(* CODESYS project TrabalhoFinal.project

Project tree, tasks and I/O mapping:
  Device : CODESYS Control Win V3, 3S - Smart Software Solutions GmbH, order no. 305021, version 3.5.11.30
    application Application
      libraries: Standard, * (System); Util, * (System)
      task MainTask (cyclic, interval t#20ms, priority 1) calls PLC_PRG
      program PLC_PRG [LD]
      Symbols
*)

// Device/Application/PLC_PRG
PROGRAM PLC_PRG
VAR
	_PassaCaixa: BOOL;
	_AtBack:BOOL;
	_AtEntry:BOOL;
	_AtFront:BOOL;
	_AtLeftEntry:BOOL;
	_AtLeftExit:BOOL;
	_AtLoadPosition:BOOL;
	_AtRigthEntry:BOOL;
	_AtRigthExit:BOOL;
	_AtTurnableEntry:BOOL;
	_AtUnloadPosition:BOOL;
	_Auto:BOOL;
	_EmergencyStop:BOOL;
	_HighBox:BOOL;
	_LowBox:BOOL;
	_Pallet:BOOL;
	_Manual:BOOL;
	_Resert:BOOL;
	_Start:BOOL;
	_Stop:BOOL;

	EntryConveyor:BOOL;
	FeederConveyor:BOOL;
	GreenIndicator:BOOL;
	LeftConveyor:BOOL;
	Load:BOOL;
	RedIndicator:BOOL;
	ResetLigth:BOOL;
	RightConveyor:BOOL;
	StartLigth:BOOL;
	StopLigth:BOOL;
	Turn:BOOL;
	Unload:BOOL;
	YellowIndicator:BOOL;
	ShortBox:BOOL;
	HighBox:BOOL;
	Trig_Right_Entry : F_TRIG;
	Trig_Left_Exit : F_TRIG;
	Trig_Rigth_Exit : F_TRIG;
	Trig_Mov1 : R_TRIG;
	Trig_Mov2 : R_TRIG;
	Trig_Mov3 : R_TRIG;
	Trig_Mov4 : R_TRIG;
	Trig_Mov5 : R_TRIG;
	Trig_turnable_Entry : F_TRIG;
	aux: INT;
	aux1:INT;
	aux2:INT;
	aux3:INT;
	auxMov1: BOOL;
	auxMov2: BOOL;
	auxMov3: BOOL;
	TON_0: TON;
	TON_1: TON;
	VarTimer1: TIME;
	VarTimer2: TIME;
	VarTimer3: TIME;
	Descarrega:BOOL;
	carregaAtivaLoad: BOOL;
	descarregaAtivaLoad: BOOL;
	descarregaAtivaUnload: BOOL;
	R_TRIG_0: R_TRIG;
	resetAux:bool;
	F_TRIG_0: F_TRIG;
	F_TRIG_1: F_TRIG;
	F_TRIG_2: F_TRIG;
	TON_2: TON;
	aux4: INT;
	ativadorTurn:BOOL;
	CTU_0: CTU;
	resetContadores: BOOL;
	contCaixasTotal:int;
	CTU_1: CTU;
	contCaixaAltas: INT;
	contCaixaBaixas: INT;
	F_TRIG_3: F_TRIG;
	F_TRIG_4: F_TRIG;
	F_TRIG_5: F_TRIG;
	
	para_esteira_principal:BOOL;
	
	sup_ligar:BOOL;
	sup_desligar:BOOL;
	sup_emergencia:BOOL;
	sup_reset:BOOL;

	sup_pos_rota:INT;
	
	
	R_TRIG_1: R_TRIG;
END_VAR
VAR // added by the converter: edge detectors and wires of the graphical bodies
    _w1, _w2, _w3, _w4, _w5 : BOOL;
END_VAR

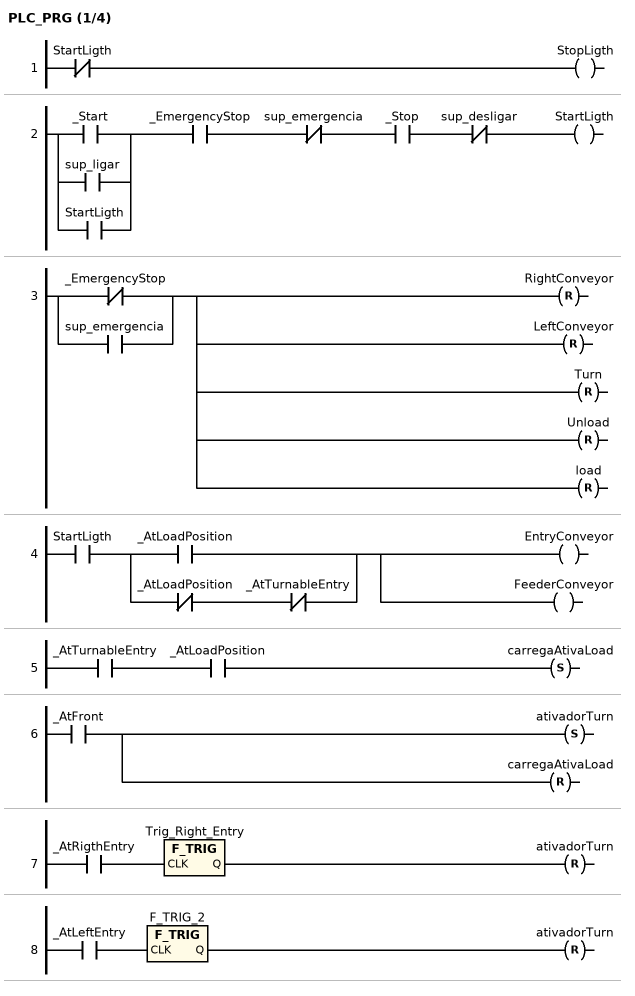
// NETWORK 1
StopLigth := NOT StartLigth;

// NETWORK 2
StartLigth := (_Start OR sup_ligar OR StartLigth) AND _EmergencyStop AND NOT sup_emergencia AND _Stop AND NOT sup_desligar;

// NETWORK 3
_w1 := NOT _EmergencyStop OR sup_emergencia;
RightConveyor R= _w1;
LeftConveyor R= _w1;
Turn R= _w1;
Unload R= _w1;
load R= _w1;

// NETWORK 4
_w2 := StartLigth AND (_AtLoadPosition OR NOT _AtLoadPosition AND NOT _AtTurnableEntry);
EntryConveyor := _w2;
FeederConveyor := _w2;

// NETWORK 5
carregaAtivaLoad S= _AtTurnableEntry AND _AtLoadPosition;

// NETWORK 6
ativadorTurn S= _AtFront;
carregaAtivaLoad R= _AtFront;

// NETWORK 7
Trig_Right_Entry(CLK := _AtRigthEntry); // F_TRIG
ativadorTurn R= Trig_Right_Entry.Q;

// NETWORK 8
F_TRIG_2(CLK := _AtLeftEntry); // F_TRIG
ativadorTurn R= F_TRIG_2.Q;

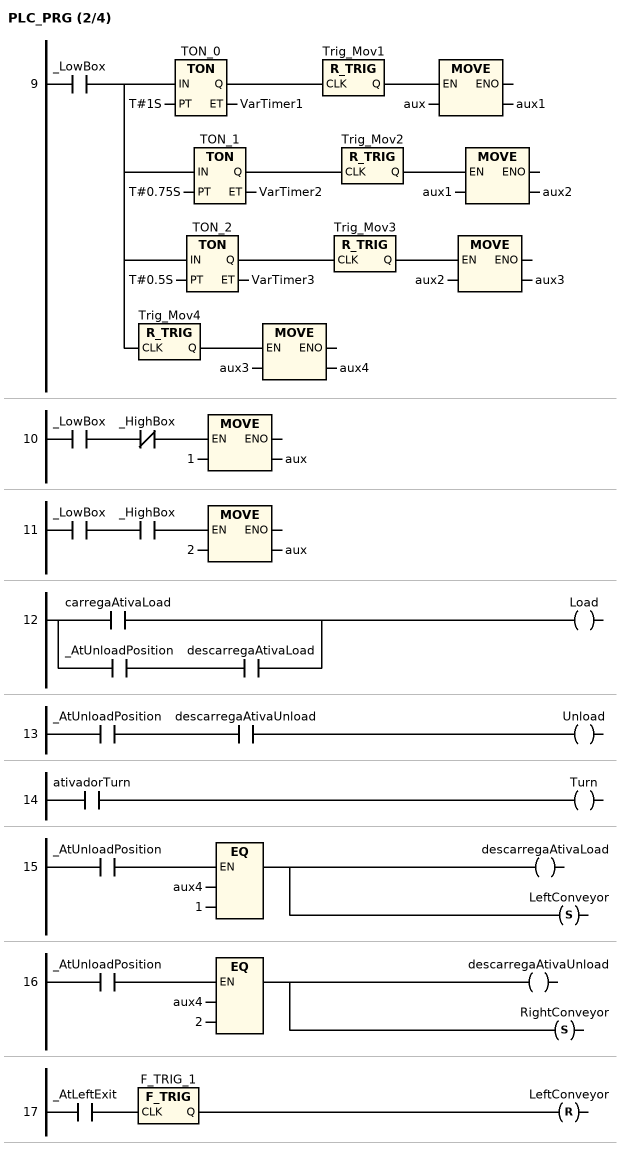
// NETWORK 9
TON_0(IN := _LowBox, PT := T#1S, ET => VarTimer1); // TON
Trig_Mov1(CLK := TON_0.Q); // R_TRIG
IF Trig_Mov1.Q THEN aux1 := aux; END_IF
TON_1(IN := _LowBox, PT := T#0.75S, ET => VarTimer2); // TON
Trig_Mov2(CLK := TON_1.Q); // R_TRIG
IF Trig_Mov2.Q THEN aux2 := aux1; END_IF
TON_2(IN := _LowBox, PT := T#0.5S, ET => VarTimer3); // TON
Trig_Mov3(CLK := TON_2.Q); // R_TRIG
IF Trig_Mov3.Q THEN aux3 := aux2; END_IF
Trig_Mov4(CLK := _LowBox); // R_TRIG
IF Trig_Mov4.Q THEN aux4 := aux3; END_IF

// NETWORK 10
IF _LowBox AND NOT _HighBox THEN aux := 1; END_IF

// NETWORK 11
IF _LowBox AND _HighBox THEN aux := 2; END_IF

// NETWORK 12
Load := carregaAtivaLoad OR _AtUnloadPosition AND descarregaAtivaLoad;

// NETWORK 13
Unload := _AtUnloadPosition AND descarregaAtivaUnload;

// NETWORK 14
Turn := ativadorTurn;

// NETWORK 15
_w3 := _AtUnloadPosition AND aux4 = 1;
descarregaAtivaLoad := _w3;
LeftConveyor S= _w3;

// NETWORK 16
_w4 := _AtUnloadPosition AND aux4 = 2;
descarregaAtivaUnload := _w4;
RightConveyor S= _w4;

// NETWORK 17
F_TRIG_1(CLK := _AtLeftExit); // F_TRIG
LeftConveyor R= F_TRIG_1.Q;

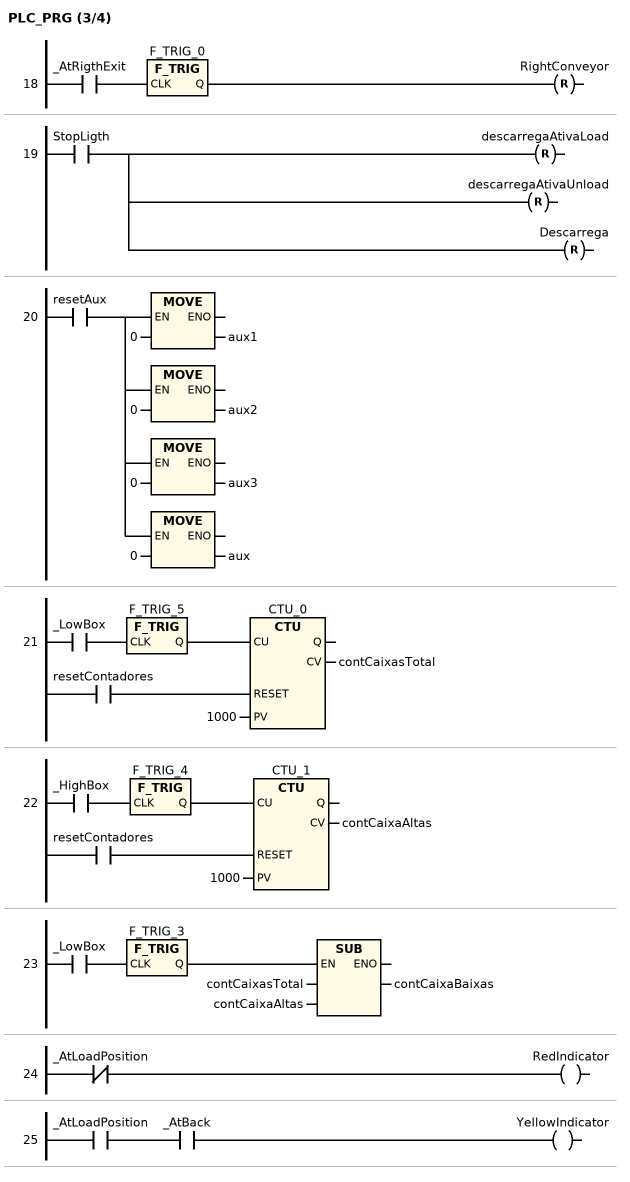
// NETWORK 18
F_TRIG_0(CLK := _AtRigthExit); // F_TRIG
RightConveyor R= F_TRIG_0.Q;

// NETWORK 19
descarregaAtivaLoad R= StopLigth;
descarregaAtivaUnload R= StopLigth;
Descarrega R= StopLigth;

// NETWORK 20
IF resetAux THEN aux1 := 0; END_IF
IF resetAux THEN aux2 := 0; END_IF
IF resetAux THEN aux3 := 0; END_IF
IF resetAux THEN aux := 0; END_IF

// NETWORK 21
F_TRIG_5(CLK := _LowBox); // F_TRIG
CTU_0(CU := F_TRIG_5.Q, RESET := resetContadores, PV := 1000, CV => contCaixasTotal); // CTU

// NETWORK 22
F_TRIG_4(CLK := _HighBox); // F_TRIG
CTU_1(CU := F_TRIG_4.Q, RESET := resetContadores, PV := 1000, CV => contCaixaAltas); // CTU

// NETWORK 23
F_TRIG_3(CLK := _LowBox); // F_TRIG
IF F_TRIG_3.Q THEN contCaixaBaixas := contCaixasTotal - contCaixaAltas; END_IF

// NETWORK 24
RedIndicator := NOT _AtLoadPosition;

// NETWORK 25
YellowIndicator := _AtLoadPosition AND _AtBack;

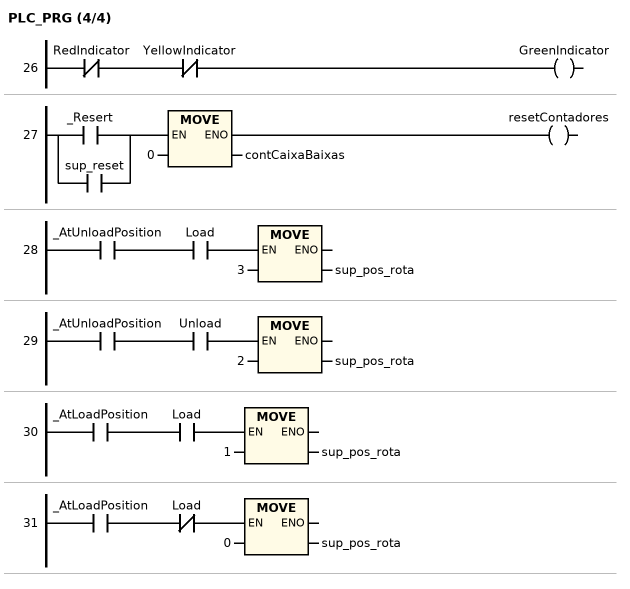
// NETWORK 26
GreenIndicator := NOT RedIndicator AND NOT YellowIndicator;

// NETWORK 27
_w5 := _Resert OR sup_reset;
IF _w5 THEN contCaixaBaixas := 0; END_IF
resetContadores := _w5;

// NETWORK 28
IF _AtUnloadPosition AND Load THEN sup_pos_rota := 3; END_IF

// NETWORK 29
IF _AtUnloadPosition AND Unload THEN sup_pos_rota := 2; END_IF

// NETWORK 30
IF _AtLoadPosition AND Load THEN sup_pos_rota := 1; END_IF

// NETWORK 31
IF _AtLoadPosition AND NOT Load THEN sup_pos_rota := 0; END_IF

END_PROGRAM
